PROGRAM MAIN
VAR
    fbTestSuite : FB_TcUnitSuite;
END_VAR

TcUnit.RUN();

END_PROGRAM

(* stored: Version 1.1.0.1, ProductVersion 3.1.4022.12
   POU MAIN: Id {aa895dfd-fdfd-4d89-a7a5-c8f63969d434}, SpecialFunc None *)
